TYPE ST_DebugSensors_SideshiftEmulation :
STRUCT
	EnableSensorDebug	: BOOL; 					// Overwrite sensor values with debug sensor values
	HW_Inputs			: ST_HW_InputsSideshift;	// Debug sensors
END_STRUCT
END_TYPE

(* stored: Version 1.1.0.1, ProductVersion 3.1.4024.9
   DUT ST_DebugSensors_SideshiftEmulation: Id {2af8dee7-02a4-4c9d-9d9b-406ab71c6176} *)
